(* Logix 5000 project; controller IsaacExample 1769-L16ER-BB1B rev 32.11; software revision 32.00 *)

TASK MainTask (continuous, watchdog 500 ms) : MainProgram, Isaac_Interface

MODULES
   Local : 1769-L16ER-BB1B (PointIO 0, rev 32.11)
      Isaac_1 : ETHERNET-MODULE (Ethernet 192.168.2.101, rev 1.1, Output RPI 20 ms)
      Isaac_2 : ETHERNET-MODULE (Ethernet 192.168.2.102, rev 1.1, Output RPI 20 ms)
      Isaac_0 : ETHERNET-MODULE (Ethernet 192.168.2.100, rev 1.1, Output RPI 20 ms)
           Isaac_0:C.Data[0]   // StartMode
           Isaac_0:C.Data[1]   // Current Program
           Isaac_0:C.Data[2]   // Results Out
           Isaac_0:C.Data[3]   // Results Out Fraction
           Isaac_0:C.Data[4]   // Baud Rate
           Isaac_0:C.Data[5]   // Data Logging
           Isaac_0:C.Data[6]   // Pressure Units
           Isaac_0:C.Data[7]   // Flow Units
           Isaac_0:C.Data[8]   // Test Pressure Digits
           Isaac_0:C.Data[10]   // Flow Digits
           Isaac_0:C.Data[9]   // Results Pressure Digits
           Isaac_0:C.Data[11]   // Spare1
           Isaac_0:C.Data[12]   // CosType-LSB
           Isaac_0:C.Data[13]   // CosType-MSB
           Isaac_0:C.Data[14]   // Spare2
           Isaac_0:C.Data[15]   // Spare3
      Isaac_3 : ETHERNET-MODULE (Ethernet 192.168.2.103, rev 1.1, Output RPI 20 ms)
      Discrete_IO : Embedded (PointIO 1, rev 32.11, Output RPI 20 ms)
           Local:1:I.Data.1   // Red Push Btn
           Local:1:I.Data.2   // 2nd Green Btn
           Local:1:I.Data.0   // Green Btn
END_MODULES

TYPE IsaacCfg :
STRUCT
   AntiTie : SINT;   // AntiTie
   CurrentProgram : SINT;   // CurrentProgram
   ResultsOut : SINT;   // Results Out
   ResultsOutFraction : SINT;   // Results Out Fraction
   BaudRate : SINT;   // Baud Rate
   DataLogging : SINT;   // Data Logging
   PressureUnits : SINT;   // Pressure Units
   FlowUnits : SINT;   // Flow Units
   TestPresDigits : SINT;   // Test Pressure Digits
   ResultsPresDigits : SINT;   // Results Pressure Digits
   FlowPressureDigits : SINT;   // Flow Pressure Digits
   SpareCfg1 : SINT;   // SpareCfg1
   cosType : INT;   // ChangeOfState flags
   SpareCfg2 : SINT;   // SpareCfg2
   SpareCfg3 : SINT;   // SpareCfg3
END_STRUCT
END_TYPE

TYPE IsaacFirmwareCfg :
STRUCT
   CosType : INT;   // ChangeOfState Type
   ClassId : INT;   // ClassId
   Instance : INT;   // Instance
   Attribute : INT;   // Attribute
   LockPrgEdits : BOOL;   // LockPrgEdits
   LockCurrentPrgEdits : BOOL;   // LockCurrentPrgEdits
   LockCalibrationEdits : BOOL;   // LockCalibrationEdit
   ElectronicReg : BOOL;   // ElectronicReg
   ManualReg : BOOL;   // ManualReg
   Concurrent : BOOL;   // Concurrent
   BuzzerEnabled : BOOL;   // BuzzerEnabled
   BusyImm : BOOL;   // BusyImm
   DhcpEnabled : BOOL;   // DhcpEnabled
   OkToResetDevice : BOOL;   // OkToResetDevice
   LinkedFail : BOOL;   // LinkedFail
   HighBleed : BOOL;   // HighBleed
   ElectRegAlwaysOn : BOOL;   // ElectRegAlwaysOn
   SpareBit13 : BOOL;   // SpareBit_12
   SpareBit14 : BOOL;   // SpareBit_13
   SpareBit15 : BOOL;   // SpareBit_14
   TesterNumber : SINT;   // TesterNumber
   BaudRate : SINT;   // BaudRate
   DataLogging : SINT;   // DataLogging
   PressureUnits : SINT;   // PressUnts
   FlowUnits : SINT;   // FlowUnts
   TestPresDigits : SINT;   // TestDigits
   ResultsPresDigits : SINT;   // ResultsDigits
   FlowPresDigits : SINT;   // FlowDigits
   BCD : SINT;   // BCD
   NumberChannels : SINT;   // NumChans
   Sensors : SINT;   // Sensors
   AntiTie : SINT;   // LockedFlgs
   AvailTestTypes : SINT;   // AvailTestTypes
   SpareByte1 : SINT;   // SpareByte1
   SpareInt1 : INT;   // SpareInt1
   IoResetTime : INT;   // IoRstTime
   FilterPress : DINT;   // FilterPress
   FilterFlow : DINT;   // FilterFlow
   FilterFillSettle : DINT;   // FilterFillSettle
   FilterElectReg : DINT;   // FilterElectReg
   HighBleedPressure : INT;   // HighBleedPres
   SpareInt2 : INT;   // SpareInt2
   AtmPress : DINT;   // AtmPress
   SerialNumber : STRING_16;   // SerialNbr
   IpAddress : STRING_16;   // IpAddr
   IpNetmask : STRING_16;   // IpNetmask
   IpGateway : STRING_16;   // ipGateway
   MacAddress : STRING_20;   // MacAddr
   DateTime : STRING_20;   // DateTime
   ModelNumber : STRING_24;   // ModelNumber
   OptionsAndFittings : STRING_32;   // OptionsAndFittings
   SccsRevDate : STRING_24;   // SccsRevDate
   SccsRev : STRING_12;   // SccsRev
   SccsRevRange : STRING_24;   // SccsRevRange
END_STRUCT
END_TYPE

TYPE IsaacIN :
STRUCT
   CosStatus : BOOL;   // Status Changed
   CosSequencePts : BOOL;   // Test Sequence Point
   CosTestStart : BOOL;   // Test has started
   CosTestResults : BOOL;   // Test has completed
   CosPressure : BOOL;   // Pressure change and not testing
   CosProgram : BOOL;   // Program parameters have changed
   CosFirmwareCfg : BOOL;   // Firmware parameters have changed
   CosProgNumb : BOOL;   // Current Program number changed
   CosTestValve : BOOL;   // Test pressure value open/closed
   SpareBit9 : BOOL;
   ClassId : INT;   // ClassId
   Instance : INT;   // Instance
   Attribute : INT;   // Attribute
   Busy : BOOL;   // Busy
   GlobalPass : BOOL;   // All Ports pass
   GlobalFail : BOOL;   // One or more ports failed
   Fail_1 : BOOL;   // Port 1 failed
   Fail_2 : BOOL;   // Port 2 failed
   Fail_3 : BOOL;   // Port 3 failed
   Fail_4 : BOOL;   // Port 4 failed
   Pass_1 : BOOL;   // Port 1 passed
   Pass_2 : BOOL;   // Port 2 passed
   Pass_3 : BOOL;   // Port 3 passed
   Pass_4 : BOOL;   // Port 4 passed
   AntiTie : BOOL;   // AntiTie Enabled
   Interlock : BOOL;   // Interlock Enabled
   Abort : BOOL;   // Abort
   SpareBit14 : BOOL;   // SpareBit14
   Fault : BOOL;   // Fault
   SpareBit16 : BOOL;   // SpareBit16
   SpareBit17 : BOOL;   // SpareBit17
   SpareBit18 : BOOL;   // SpareBit18
   SpareBit19 : BOOL;   // SpareBit19
   SpareBit20 : BOOL;   // SpareBit20
   SpareBit21 : BOOL;   // SpareBit21
   SpareBit22 : BOOL;   // SpareBit22
   SpareBit23 : BOOL;   // SpareBit23
   SpareBit24 : BOOL;   // SpareBit24
   SpareBit25 : BOOL;   // SpareBit25
   SpareBit26 : BOOL;   // SpareBit26
   SpareBit27 : BOOL;   // SpareBit27
   SpareBit28 : BOOL;   // SpareBit28
   SpareBit29 : BOOL;   // SpareBit29
   SpareBit30 : BOOL;   // SpareBit30
   SpareBit31 : BOOL;   // SpareBit31
   SpareByteIn1 : SINT;   // SpareByteIn1
   TestPresValve1 : BOOL;   // TestPresValve1
   TestPresValve2 : BOOL;   // TestPresValve2
   TestPresValve3 : BOOL;   // TestPresValve3
   TestPresValve4 : BOOL;   // TestPresValve4
   CurrentProgram : SINT;   // CurrentProgram
   TestType : SINT;   // Type of test running
   PortEnabled1 : BOOL;   // PortEnabled1
   PortEnabled2 : BOOL;   // PortEnabled2
   PortEnabled3 : BOOL;   // PortEnabled3
   PortEnabled4 : BOOL;   // PortEnabled4
   Sequence : SINT;   // Sequence
   SpareIntIn1 : INT;   // SpareIntIn1
   ElapseTime : DINT;   // ElapseTime
   PortStatus1 : SINT;   // PortStatus1
   PortStatus2 : SINT;   // PortStatus2
   PortStatus3 : SINT;   // PortStatus3
   PortStatus4 : SINT;   // PortStatus4
   PressurePort1 : DINT;   // Test Pressure at port 1
   PressurePort2 : DINT;   // Test Pressure at port 2
   PressurePort3 : DINT;   // Test Pressure at port 3
   PressurePort4 : DINT;   // Test Pressure at port 4
   TestResults1 : DINT;   // TestResults1
   TestResults2 : DINT;   // TestResults2
   TestResults3 : DINT;   // TestResults3
   TestResults4 : DINT;   // TestResults4
   Flow : DINT;   // Flow
   SpareDIntIn1 : DINT;   // SpareDIntIn1
END_STRUCT
END_TYPE

TYPE IsaacOUT :
STRUCT
   Start : BOOL;   // Start
   StartAntiTie : BOOL;   // StartAntiTie
   Abort : BOOL;   // Abort
   Retest : BOOL;   // Retest
   Valve1On : BOOL;   // Valve1On
   Valve2On : BOOL;   // Valve2On
   Valve3On : BOOL;   // Valve3On
   Valve4On : BOOL;   // Valve4On
   IgnoreCmds : BOOL;   // IgnoreCmds
   StatusGet : BOOL;   // StatusGet
   SpareBit10 : BOOL;   // SpareBit10
   SpareBit11 : BOOL;   // SpareBit11
   SpareBit12 : BOOL;   // SpareBit12
   SpareBit13 : BOOL;   // SpareBit13
   SpareBit14 : BOOL;   // SpareBit14
   SpareBit15 : BOOL;   // SpareBit15
   SpareBit16 : BOOL;   // SpareBit16
   SpareBit17 : BOOL;   // SpareBit17
   SpareBit18 : BOOL;   // SpareBit18
   SpareBit19 : BOOL;   // SpareBit19
   SpareBit20 : BOOL;   // SpareBit20
   SpareBit21 : BOOL;   // SpareBit21
   SpareBit22 : BOOL;   // SpareBit22
   SpareBit23 : BOOL;   // SpareBit23
   SpareBit24 : BOOL;   // SpareBit24
   SpareBit25 : BOOL;   // SpareBit25
   SpareBit26 : BOOL;   // SpareBit26
   SpareBit27 : BOOL;   // SpareBit27
   SpareBit28 : BOOL;   // SpareBit28
   SpareBit29 : BOOL;   // SpareBit29
   SpareBit30 : BOOL;   // SpareBit30
   SpareBit31 : BOOL;   // SpareBit31
   CurrentProgram : SINT;   // CurrentProgram
   SpareByteOut1 : SINT;   // SpareByteOut1
   SpareIntOut1 : INT;   // SpareIntOut1
   SpareDIntOut1 : DINT;   // SpareDIntOut1
   SpareDIntOut2 : DINT;   // SpareDIntOut2
END_STRUCT
END_TYPE

TYPE IsaacProgram :
STRUCT
   CosType : INT;   // ChangeOfState Type
   ClassId : INT;   // ClassId
   Instance : INT;   // Instance
   Attribute : INT;   // Attribute
   PrgNumb : SINT;   // PrgNumb
   SpareByte1 : SINT;   // SpareByte1
   Loops : INT;   // Loops
   PortEnabled1 : BOOL;   // PortEnabled1
   PortEnabled2 : BOOL;   // PortEnabled2
   PortEnabled3 : BOOL;   // PortEnabled3
   PortEnabled4 : BOOL;   // PortEnabled4
   FixtureValve1 : BOOL;   // FixtureValve1
   FixtureValve2 : BOOL;   // FixtureValve2
   ClampHoldFail : BOOL;   // ClampHoldFail
   Rslts232 : BOOL;   // Rslts232
   RsltsEthr : BOOL;   // RsltsEthr
   AutoFFill : BOOL;   // AutoFFill
   LeakStd : BOOL;   // LeakStd
   AutoVent : BOOL;   // AutoVent
   IncreaseLimit : BOOL;   // IncLimitEnbl
   EvalAtEnd : BOOL;   // EvalAtEnd
   ElectReg : BOOL;   // ElectReg
   SpareBit_15 : BOOL;   // SpareBit_15
   SpareBit_16 : BOOL;   // SpareBit_16
   SpareBit_17 : BOOL;   // SpareBit_17
   SpareBit_18 : BOOL;   // SpareBit_18
   SpareBit_19 : BOOL;   // SpareBit_19
   SpareBit_20 : BOOL;   // SpareBit_20
   SpareBit_21 : BOOL;   // SpareBit_21
   SpareBit_22 : BOOL;   // SpareBit_22
   SpareBit_23 : BOOL;   // SpareBit_23
   SpareBit_24 : BOOL;   // SpareBit_24
   SpareBit_25 : BOOL;   // SpareBit_25
   SpareBit_26 : BOOL;   // SpareBit_26
   SpareBit_27 : BOOL;   // SpareBit_27
   SpareBit_28 : BOOL;   // SpareBit_28
   SpareBit_29 : BOOL;   // SpareBit_29
   SpareBit_30 : BOOL;   // SpareBit_30
   SpareBit_31 : BOOL;   // SpareBit_31
   TestType : SINT;   // TestType
   NextPrg : SINT;   // NextPrg
   ElectRegDelay : SINT;   // ElectRegDelay
   SpareByte2 : SINT;   // SpareByte2
   TimeIdle : DINT;   // TimeIdle
   TimeClmp1 : DINT;   // TimeClmp1
   TimeClmp2 : DINT;   // TimeClmp2
   TimeFFill : DINT;   // TimeFFill
   TimeFill : DINT;   // TimeFill
   TimeSettle : DINT;   // TimeSettle
   TimeTest : DINT;   // TimeTest
   TimeVent : DINT;   // TimeVent
   TimeUnClmp1 : DINT;   // TimeUnClmp1
   TimeUnClmp2 : DINT;   // TimeUnClmp2
   SpareDInt1 : DINT;   // SpareDInt_1
   SpareDInt2 : DINT;   // SpareDInt_2
   TestPres : DINT;   // TestPres
   TestPresMin : DINT;   // RestPresMin
   TestPresMax : DINT;   // TestPresMax
   RegKp : DINT;   // RegKP
   RegKi : DINT;   // RegKi
   RegKd : DINT;   // RegKd
   PresFFill : DINT;   // PresFFill
   PresTestMin : DINT;   // PresTestMin
   PresTestMax : DINT;   // PresTestMax
   PresTestTrigger : DINT;   // PresTestTrigger
   Volume : DINT;   // Volume
   RampRate : DINT;   // RampRate
   SpareDInt3 : DINT;   // SpareDInt_3
   PrgName : STRING_16;   // PrgName
END_STRUCT
END_TYPE

TYPE STRING_12 :
STRUCT
   LEN : DINT;
   DATA : SINT[12];
END_STRUCT
END_TYPE

TYPE STRING_16 :
STRUCT
   LEN : DINT;
   DATA : SINT[16];
END_STRUCT
END_TYPE

TYPE STRING_20 :
STRUCT
   LEN : DINT;
   DATA : SINT[20];
END_STRUCT
END_TYPE

TYPE STRING_24 :
STRUCT
   LEN : DINT;
   DATA : SINT[24];
END_STRUCT
END_TYPE

TYPE STRING_32 :
STRUCT
   LEN : DINT;
   DATA : SINT[32];
END_STRUCT
END_TYPE

ADD_ON_INSTRUCTION Isaac_Run   (* revision 1.0, vendor Zaxis, Inc *)
// Start Test
VAR_INPUT
   Start : BOOL; {access Read Only, required}   // Test Start
   AntiTie : BOOL; {access Read Only, required}   // AntiTie Bit
   AbortTest : BOOL; {access Read Only, required}   // Abort Bit
END_VAR
VAR_IN_OUT
   IT : IsaacTester; {required}
END_VAR

ROUTINE Logic   (* ladder *)
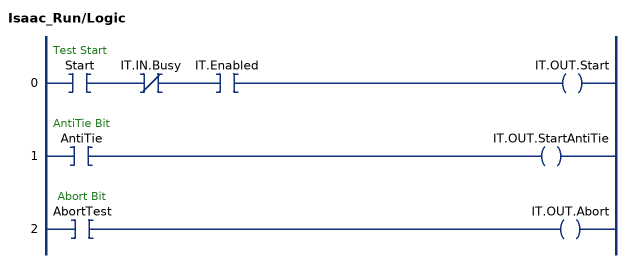
   0: XIC(Start)XIO(IT.IN.Busy)XIC(IT.Enabled)OTE(IT.OUT.Start);
   1: XIC(AntiTie)OTE(IT.OUT.StartAntiTie);
   2: XIC(AbortTest)OTE(IT.OUT.Abort);
END_ROUTINE
END_ADD_ON_INSTRUCTION

VAR_GLOBAL   (* controller tags *)
   Button_AntiTie : ALIAS FOR Local:1:I.Data.2;
   Button_Start : ALIAS FOR Local:1:I.Data.0;
   Button_Stop : ALIAS FOR Local:1:I.Data.1;
   Isaac_Testers : IsaacTester[4] := ([0].Enabled := 1, [0].IpAddress := '$0D192.168.2.10', [0].PathToEthMod := '$00$12$0D192.168.2.10', [0].PathToGSVModule := '$10$00$12$0D192.168.2.100', [0].IN.ClassId := 104, [0].IN.Attribute := 6, [0].IN.GlobalPass := 1, [0].IN.Pass_1 := 1, [0].IN.PortEnabled1 := 1, [0].IN.Sequence := 6, [0].IN.ElapseTime := 48, [0].IN.PortStatus1 := -1, [0].IN.PressurePort1 := 560, [0].IN.TestResults1 := 847, [1].Enabled := 1, [2].Enabled := 1, [3].Enabled := 1);
   IsaacFirmware : IsaacFirmwareCfg;
   IsaacFirmware_Read : MESSAGE;
        MessageParameters(ServiceCode := 16#0001, DestinationTag := IsaacFirmware, ...)
   IsaacFirmware_Write : MESSAGE;
        .UnconnectedTimeout   // Timeout down to 3 seconds
        MessageParameters(ServiceCode := 16#0002, LocalElement := IsaacFirmware, ...)
   IsaacProgram : IsaacProgram;
   IsaacProgram_Read : MESSAGE;
        MessageParameters(ServiceCode := 16#0001, DestinationTag := IsaacProgram, ...)
   IsaacProgram_Write : MESSAGE;
        MessageParameters(ServiceCode := 16#0002, LocalElement := IsaacProgram, ...)
END_VAR

PROGRAM Isaac_Interface   (* main routine Isaac_Run *)
VAR
   Firmware_Read : BOOL;
   Firmware_Write : BOOL;
   Program_Read : BOOL;
   Program_Write : BOOL;
   Run_Enabled : BOOL := 1;
   StartTest : Isaac_Run;
END_VAR

ROUTINE Isaac_MapInputs   (* ladder *)
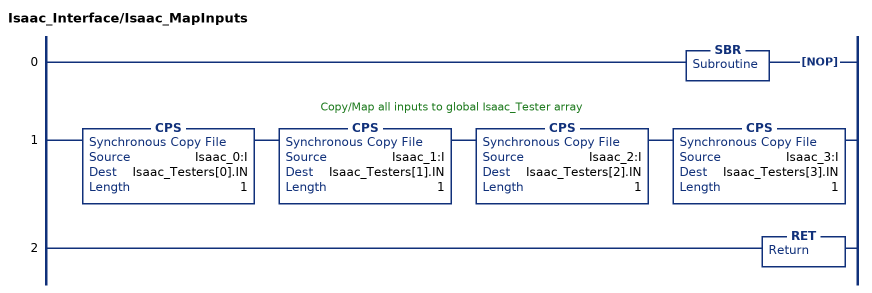
   0: SBR()NOP();
   // Copy/Map all inputs to global Isaac_Tester array
   1: CPS(Isaac_0:I,Isaac_Testers[0].IN,1)CPS(Isaac_1:I,Isaac_Testers[1].IN,1)CPS(Isaac_2:I,Isaac_Testers[2].IN,1)CPS(Isaac_3:I,Isaac_Testers[3].IN,1);
   2: RET();
END_ROUTINE

ROUTINE Isaac_MapOutputs   (* ladder *)
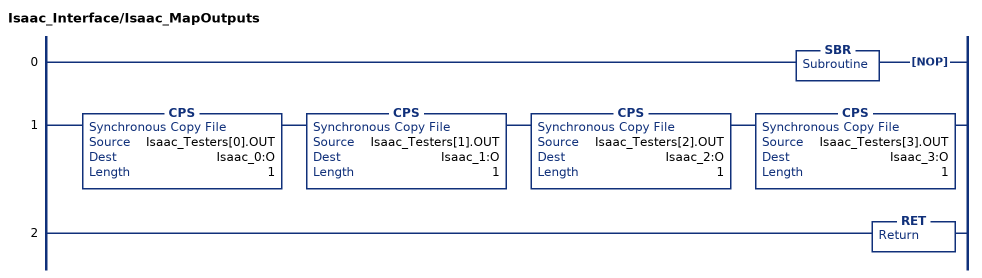
   0: SBR()NOP();
   1: CPS(Isaac_Testers[0].OUT,Isaac_0:O,1)CPS(Isaac_Testers[1].OUT,Isaac_1:O,1)CPS(Isaac_Testers[2].OUT,Isaac_2:O,1)CPS(Isaac_Testers[3].OUT,Isaac_3:O,1);
   2: RET();
END_ROUTINE

ROUTINE Isaac_Run   (* ladder *)
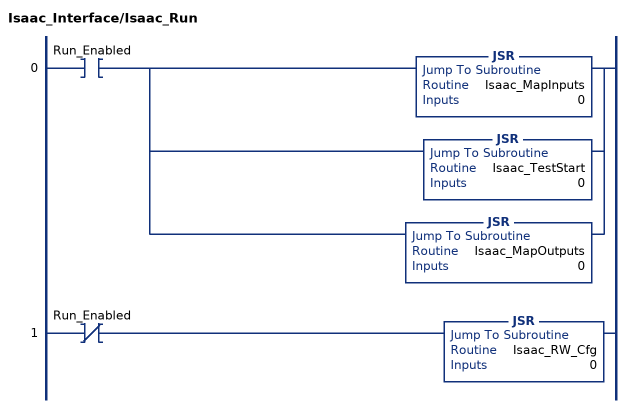
   0: XIC(Run_Enabled)[JSR(Isaac_MapInputs,0) ,JSR(Isaac_TestStart,0) ,JSR(Isaac_MapOutputs,0) ];
   1: XIO(Run_Enabled)JSR(Isaac_RW_Cfg,0);
END_ROUTINE

ROUTINE Isaac_RW_Cfg   (* ladder *)
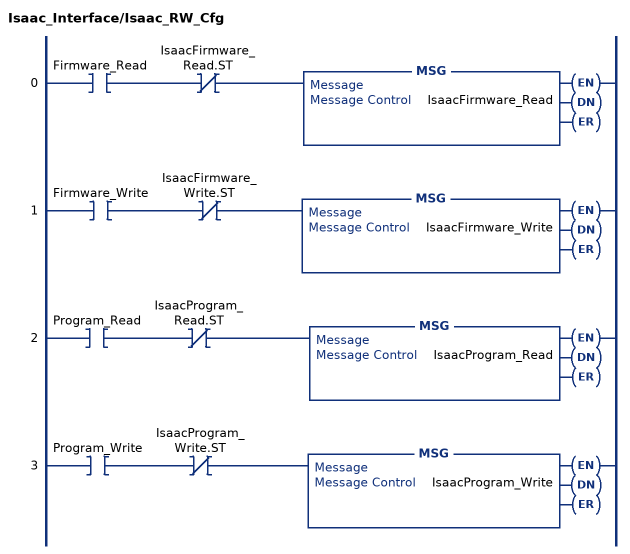
   0: XIC(Firmware_Read)XIO(IsaacFirmware_Read.ST)MSG(IsaacFirmware_Read);
   1: XIC(Firmware_Write)XIO(IsaacFirmware_Write.ST)MSG(IsaacFirmware_Write);
   2: XIC(Program_Read)XIO(IsaacProgram_Read.ST)MSG(IsaacProgram_Read);
   3: XIC(Program_Write)XIO(IsaacProgram_Write.ST)MSG(IsaacProgram_Write);
END_ROUTINE

ROUTINE Isaac_TestStart   (* ladder *)
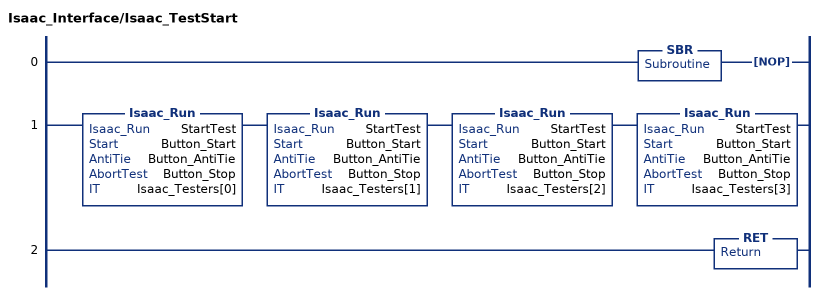
   0: SBR()NOP();
   1: Isaac_Run(StartTest,Button_Start,Button_AntiTie,Button_Stop,Isaac_Testers[0])Isaac_Run(StartTest,Button_Start,Button_AntiTie,Button_Stop,Isaac_Testers[1])Isaac_Run(StartTest,Button_Start,Button_AntiTie,Button_Stop,Isaac_Testers[2])Isaac_Run(StartTest,Button_Start,Button_AntiTie,Button_Stop,Isaac_Testers[3]);
   2: RET();
END_ROUTINE
END_PROGRAM

PROGRAM MainProgram   (* main routine MainRoutine *)

ROUTINE MainRoutine   (* ladder *)
END_ROUTINE
END_PROGRAM
